// TIA Portal project "TPP" (V16)

(* hardware
DEVICE "S7300/ET200M station_1"  S7-300 station
   slot 0: "Rail_0"  Rail  6ES7 390-1***0-0AA0
   slot 2: "PLC_1"  CPU 314C-2 PN/DP  6ES7 314-6EH04-0AB0  V3.3
      slot 2: "PROFINET interface_1"  PN-IO
         slot 1: "Port_1"  Port
         slot 2: "Port_2"  Port
      slot 5: "DI 24/DO 16_1"  DI24/DO16
      slot 6: "AI 5/AO 2_1"  AI5/AO2
      slot 7: "Count_1"  Counter
      slot 8: "Positioning_1"  Positioning
DEVICE "HMI_1"  KTP1000 Basic color PN
   slot 0: "HMI_1"  KTP1000 Basic color PN  6AV6 647-0AF11-3AX0  12.0.0.0
   slot 1: "HMI_RT_1"  KTP1000 Basic color PN  6AV6 647-0AF11-3AX0  12.0.0.0
   slot 5: "HMI_1.IE_CP_1"  PROFINET Interface  12.0.0.0
      slot 1: "Interface PROFINET_1"  PROFINET Interface
         slot 1: "Port_1"  Port
*)

// ===== PLC "PLC_1"  CPU 314C-2 PN/DP =====

VAR_GLOBAL   // PLC tag table "Default tag table"
   "DE" AT %I0.1 : Bool;
   "PP" AT %I0.2 : Bool;
   "CS" AT %I0.3 : Bool;
   "AP" AT %I0.4 : Bool;
   "C1" AT %M3.7 : Bool;
   "C2" AT %M4.0 : Bool;
   "C3" AT %M4.1 : Bool;
   "C4" AT %M4.2 : Bool;
   "C5" AT %M4.3 : Bool;
   "C6" AT %M4.4 : Bool;
   "C7" AT %M4.5 : Bool;
   "C8" AT %M4.6 : Bool;
   "C9" AT %M4.7 : Bool;
   "C10" AT %M5.0 : Bool;
   "PA" AT %Q0.0 : Bool;
   "PV" AT %Q0.1 : Bool;
   "CV1" AT %Q0.2 : Bool;
   "CV2" AT %Q0.3 : Bool;
   "GA" AT %Q0.4 : Bool;
   "CPH" AT %Q0.5 : Bool;
   "CPL" AT %Q0.6 : Bool;
   "B1" AT %M0.0 : Bool;
   "B2" AT %M0.1 : Bool;
   "B3" AT %M0.2 : Bool;
   "B4" AT %M0.3 : Bool;
   "B5" AT %M0.4 : Bool;
   "B6" AT %M0.5 : Bool;
   "B7" AT %M0.6 : Bool;
   "B8" AT %M0.7 : Bool;
   "B9" AT %M1.0 : Bool;
   "B10" AT %M1.1 : Bool;
   "B11" AT %M1.2 : Bool;
   "B12" AT %M1.3 : Bool;
   "B13" AT %M1.4 : Bool;
   "B14" AT %M1.5 : Bool;
   "B15" AT %M1.6 : Bool;
   "B16" AT %M1.7 : Bool;
   "B17" AT %M2.0 : Bool;
   "B18" AT %M2.1 : Bool;
   "B19" AT %M2.2 : Bool;
   "T1" AT %M2.5 : Bool;
   "T2" AT %M2.6 : Bool;
   "T3" AT %M2.7 : Bool;
   "T4" AT %M3.0 : Bool;
   "T5" AT %M3.1 : Bool;
   "T6" AT %M3.2 : Bool;
   "T7" AT %M3.3 : Bool;
   "T8" AT %M3.4 : Bool;
   "T9" AT %M3.5 : Bool;
   "T10" AT %M3.6 : Bool;
   "T11" AT %M5.1 : Bool;
   "T12" AT %M5.2 : Bool;
   "T13" AT %M5.3 : Bool;
   "T14" AT %M5.4 : Bool;
   "H1" AT %I0.5 : Bool;
   "H2" AT %I0.6 : Bool;
   "H3" AT %I0.7 : Bool;
   "H4" AT %I1.0 : Bool;
   "H5" AT %I1.1 : Bool;
   "H6" AT %I1.2 : Bool;
   "L1" AT %I1.3 : Bool;
   "L2" AT %I1.4 : Bool;
   "S" AT %I1.5 : Bool;
   "TC" AT %I1.6 : Bool;
   "AA" AT %Q0.7 : Bool;
END_VAR

ORGANIZATION_BLOCK "Main"   // OB1, LAD
TITLE = "Main Program Sweep (Cycle)"
{ S7_Optimized_Access := 'FALSE' }
VERSION : 0.1
   VAR_TEMP
      OB1_EV_CLASS : Byte;   // Bits 0-3 = 1 (Coming event), Bits 4-7 = 1 (Event class 1)
      OB1_SCAN_1 : Byte;   // 1 (Cold restart scan 1 of OB 1), 3 (Scan 2-n of OB 1)
      OB1_PRIORITY : Byte;   // Priority of OB Execution
      OB1_OB_NUMBR : Byte;   // 1 (Organization block 1, OB1)
      OB1_RESERVED_1 : Byte;   // Reserved for system
      OB1_RESERVED_2 : Byte;   // Reserved for system
      OB1_PREV_CYCLE : Int;   // Cycle time of previous OB1 scan (milliseconds)
      OB1_MIN_CYCLE : Int;   // Minimum cycle time of OB1 (milliseconds)
      OB1_MAX_CYCLE : Int;   // Maximum cycle time of OB1 (milliseconds)
      OB1_DATE_TIME : Date_And_Time;   // Date and time OB1 started
   END_VAR
BEGIN

REGION Network 1
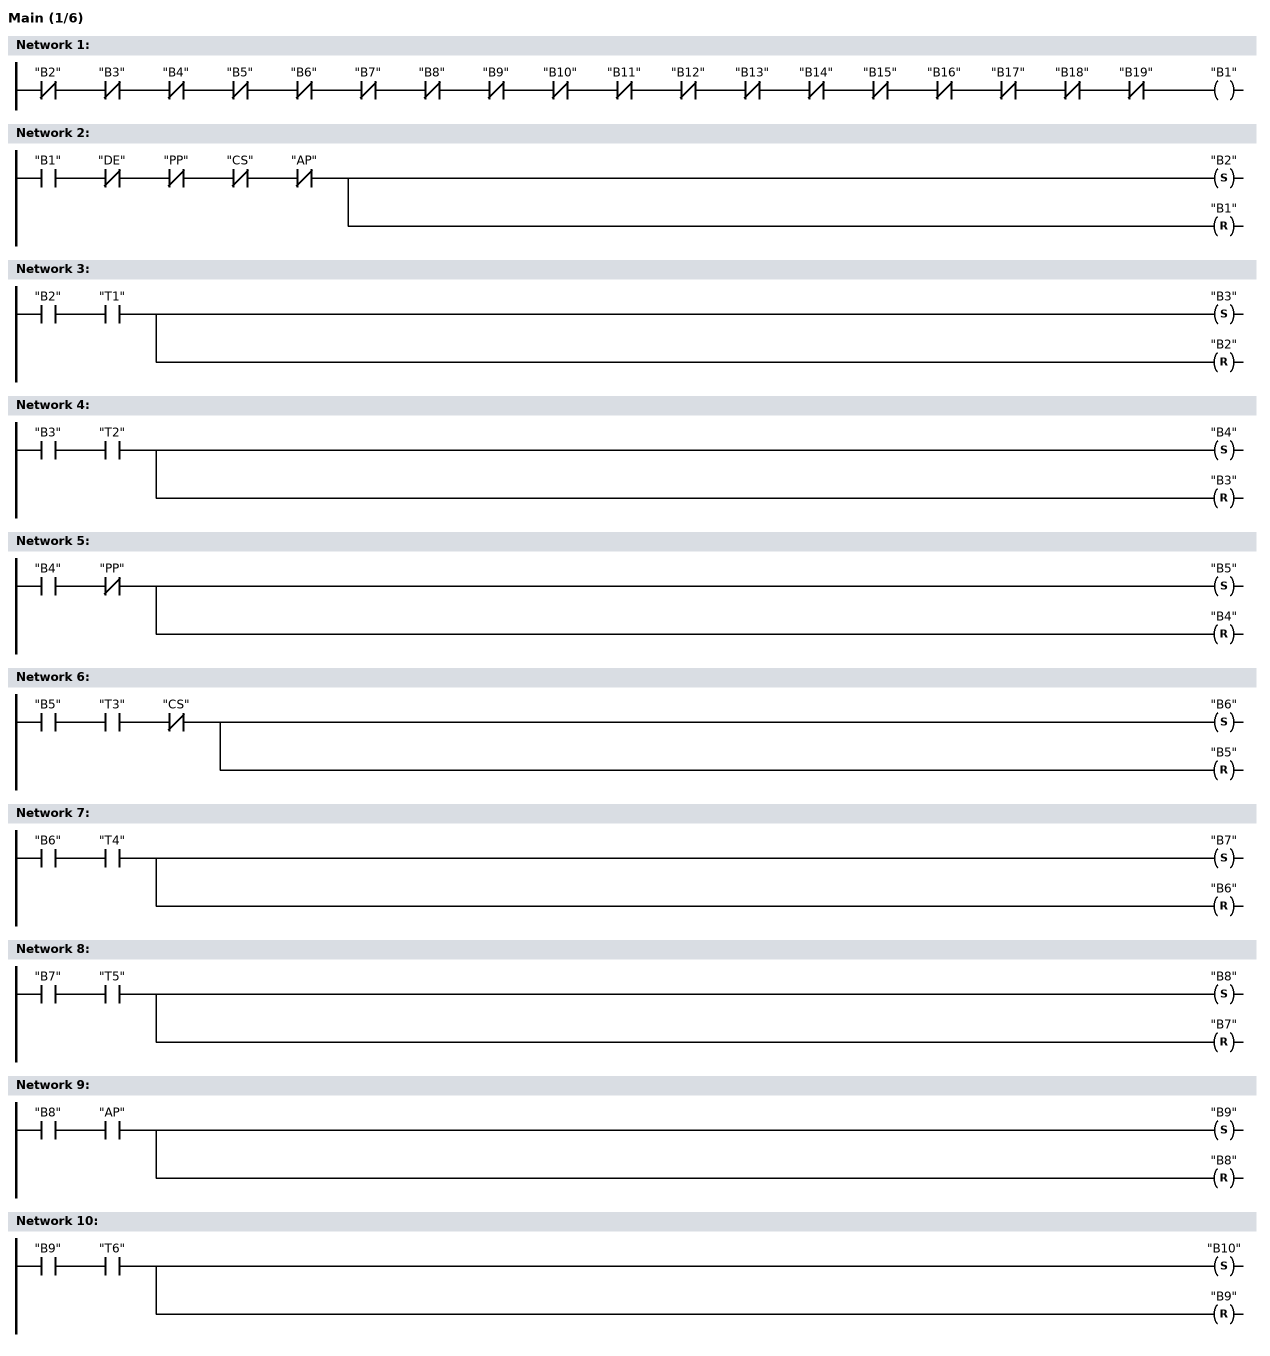
   RUNG wire#powerrail
      I_Contact( "B2" )
      I_Contact( "B3" )
      I_Contact( "B4" )
      I_Contact( "B5" )
      I_Contact( "B6" )
      I_Contact( "B7" )
      I_Contact( "B8" )
      I_Contact( "B9" )
      I_Contact( "B10" )
      I_Contact( "B11" )
      I_Contact( "B12" )
      I_Contact( "B13" )
      I_Contact( "B14" )
      I_Contact( "B15" )
      I_Contact( "B16" )
      I_Contact( "B17" )
      I_Contact( "B18" )
      I_Contact( "B19" )
      Coil( "B1" )
   END_RUNG
   // the same network as SCL:
   "B1" := NOT "B2" AND NOT "B3" AND NOT "B4" AND NOT "B5" AND NOT "B6" AND NOT "B7" AND NOT "B8" AND NOT "B9" AND NOT "B10" AND NOT "B11" AND NOT "B12" AND NOT "B13" AND NOT "B14" AND NOT "B15" AND NOT "B16" AND NOT "B17" AND NOT "B18" AND NOT "B19";
END_REGION

REGION Network 2
   RUNG wire#powerrail
      Contact( "B1" )
      I_Contact( "DE" )
      I_Contact( "PP" )
      I_Contact( "CS" )
      I_Contact( "AP" )
      wire#w1
      S_Coil( "B2" )
   END_RUNG
   RUNG wire#w1
      R_Coil( "B1" )
   END_RUNG
   // the same network as SCL:
   IF "B1" AND NOT "DE" AND NOT "PP" AND NOT "CS" AND NOT "AP" THEN
       "B2" := TRUE;
       "B1" := FALSE;
   END_IF;
END_REGION

REGION Network 3
   RUNG wire#powerrail
      Contact( "B2" )
      Contact( "T1" )
      wire#w1
      S_Coil( "B3" )
   END_RUNG
   RUNG wire#w1
      R_Coil( "B2" )
   END_RUNG
   // the same network as SCL:
   IF "B2" AND "T1" THEN
       "B3" := TRUE;
       "B2" := FALSE;
   END_IF;
END_REGION

REGION Network 4
   RUNG wire#powerrail
      Contact( "B3" )
      Contact( "T2" )
      wire#w1
      S_Coil( "B4" )
   END_RUNG
   RUNG wire#w1
      R_Coil( "B3" )
   END_RUNG
   // the same network as SCL:
   IF "B3" AND "T2" THEN
       "B4" := TRUE;
       "B3" := FALSE;
   END_IF;
END_REGION

REGION Network 5
   RUNG wire#powerrail
      Contact( "B4" )
      I_Contact( "PP" )
      wire#w1
      S_Coil( "B5" )
   END_RUNG
   RUNG wire#w1
      R_Coil( "B4" )
   END_RUNG
   // the same network as SCL:
   IF "B4" AND NOT "PP" THEN
       "B5" := TRUE;
       "B4" := FALSE;
   END_IF;
END_REGION

REGION Network 6
   RUNG wire#powerrail
      Contact( "B5" )
      Contact( "T3" )
      I_Contact( "CS" )
      wire#w1
      S_Coil( "B6" )
   END_RUNG
   RUNG wire#w1
      R_Coil( "B5" )
   END_RUNG
   // the same network as SCL:
   IF "B5" AND "T3" AND NOT "CS" THEN
       "B6" := TRUE;
       "B5" := FALSE;
   END_IF;
END_REGION

REGION Network 7
   RUNG wire#powerrail
      Contact( "B6" )
      Contact( "T4" )
      wire#w1
      S_Coil( "B7" )
   END_RUNG
   RUNG wire#w1
      R_Coil( "B6" )
   END_RUNG
   // the same network as SCL:
   IF "B6" AND "T4" THEN
       "B7" := TRUE;
       "B6" := FALSE;
   END_IF;
END_REGION

REGION Network 8
   RUNG wire#powerrail
      Contact( "B7" )
      Contact( "T5" )
      wire#w1
      S_Coil( "B8" )
   END_RUNG
   RUNG wire#w1
      R_Coil( "B7" )
   END_RUNG
   // the same network as SCL:
   IF "B7" AND "T5" THEN
       "B8" := TRUE;
       "B7" := FALSE;
   END_IF;
END_REGION

REGION Network 9
   RUNG wire#powerrail
      Contact( "B8" )
      Contact( "AP" )
      wire#w1
      S_Coil( "B9" )
   END_RUNG
   RUNG wire#w1
      R_Coil( "B8" )
   END_RUNG
   // the same network as SCL:
   IF "B8" AND "AP" THEN
       "B9" := TRUE;
       "B8" := FALSE;
   END_IF;
END_REGION

REGION Network 10
   RUNG wire#powerrail
      Contact( "B9" )
      Contact( "T6" )
      wire#w1
      S_Coil( "B10" )
   END_RUNG
   RUNG wire#w1
      R_Coil( "B9" )
   END_RUNG
   // the same network as SCL:
   IF "B9" AND "T6" THEN
       "B10" := TRUE;
       "B9" := FALSE;
   END_IF;
END_REGION

REGION Network 11
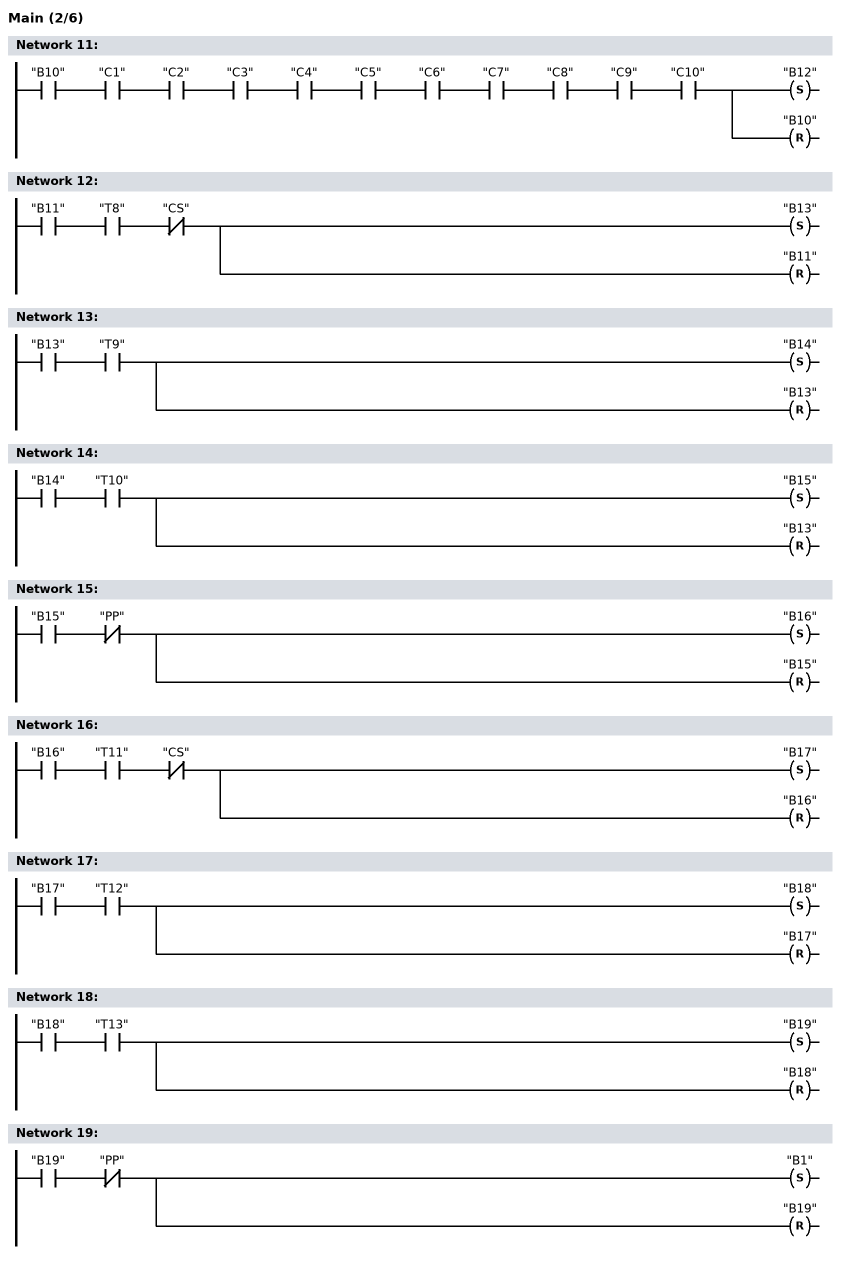
   RUNG wire#powerrail
      Contact( "B10" )
      Contact( "C1" )
      Contact( "C2" )
      Contact( "C3" )
      Contact( "C4" )
      Contact( "C5" )
      Contact( "C6" )
      Contact( "C7" )
      Contact( "C8" )
      Contact( "C9" )
      Contact( "C10" )
      wire#w1
      S_Coil( "B12" )
   END_RUNG
   RUNG wire#w1
      R_Coil( "B10" )
   END_RUNG
   // the same network as SCL:
   IF "B10" AND "C1" AND "C2" AND "C3" AND "C4" AND "C5" AND "C6" AND "C7" AND "C8" AND "C9" AND "C10" THEN
       "B12" := TRUE;
       "B10" := FALSE;
   END_IF;
END_REGION

REGION Network 12
   RUNG wire#powerrail
      Contact( "B11" )
      Contact( "T8" )
      I_Contact( "CS" )
      wire#w1
      S_Coil( "B13" )
   END_RUNG
   RUNG wire#w1
      R_Coil( "B11" )
   END_RUNG
   // the same network as SCL:
   IF "B11" AND "T8" AND NOT "CS" THEN
       "B13" := TRUE;
       "B11" := FALSE;
   END_IF;
END_REGION

REGION Network 13
   RUNG wire#powerrail
      Contact( "B13" )
      Contact( "T9" )
      wire#w1
      S_Coil( "B14" )
   END_RUNG
   RUNG wire#w1
      R_Coil( "B13" )
   END_RUNG
   // the same network as SCL:
   IF "B13" AND "T9" THEN
       "B14" := TRUE;
       "B13" := FALSE;
   END_IF;
END_REGION

REGION Network 14
   RUNG wire#powerrail
      Contact( "B14" )
      Contact( "T10" )
      wire#w1
      S_Coil( "B15" )
   END_RUNG
   RUNG wire#w1
      R_Coil( "B13" )
   END_RUNG
   // the same network as SCL:
   IF "B14" AND "T10" THEN
       "B15" := TRUE;
       "B13" := FALSE;
   END_IF;
END_REGION

REGION Network 15
   RUNG wire#powerrail
      Contact( "B15" )
      I_Contact( "PP" )
      wire#w1
      S_Coil( "B16" )
   END_RUNG
   RUNG wire#w1
      R_Coil( "B15" )
   END_RUNG
   // the same network as SCL:
   IF "B15" AND NOT "PP" THEN
       "B16" := TRUE;
       "B15" := FALSE;
   END_IF;
END_REGION

REGION Network 16
   RUNG wire#powerrail
      Contact( "B16" )
      Contact( "T11" )
      I_Contact( "CS" )
      wire#w1
      S_Coil( "B17" )
   END_RUNG
   RUNG wire#w1
      R_Coil( "B16" )
   END_RUNG
   // the same network as SCL:
   IF "B16" AND "T11" AND NOT "CS" THEN
       "B17" := TRUE;
       "B16" := FALSE;
   END_IF;
END_REGION

REGION Network 17
   RUNG wire#powerrail
      Contact( "B17" )
      Contact( "T12" )
      wire#w1
      S_Coil( "B18" )
   END_RUNG
   RUNG wire#w1
      R_Coil( "B17" )
   END_RUNG
   // the same network as SCL:
   IF "B17" AND "T12" THEN
       "B18" := TRUE;
       "B17" := FALSE;
   END_IF;
END_REGION

REGION Network 18
   RUNG wire#powerrail
      Contact( "B18" )
      Contact( "T13" )
      wire#w1
      S_Coil( "B19" )
   END_RUNG
   RUNG wire#w1
      R_Coil( "B18" )
   END_RUNG
   // the same network as SCL:
   IF "B18" AND "T13" THEN
       "B19" := TRUE;
       "B18" := FALSE;
   END_IF;
END_REGION

REGION Network 19
   RUNG wire#powerrail
      Contact( "B19" )
      I_Contact( "PP" )
      wire#w1
      S_Coil( "B1" )
   END_RUNG
   RUNG wire#w1
      R_Coil( "B19" )
   END_RUNG
   // the same network as SCL:
   IF "B19" AND NOT "PP" THEN
       "B1" := TRUE;
       "B19" := FALSE;
   END_IF;
END_REGION

REGION Network 20
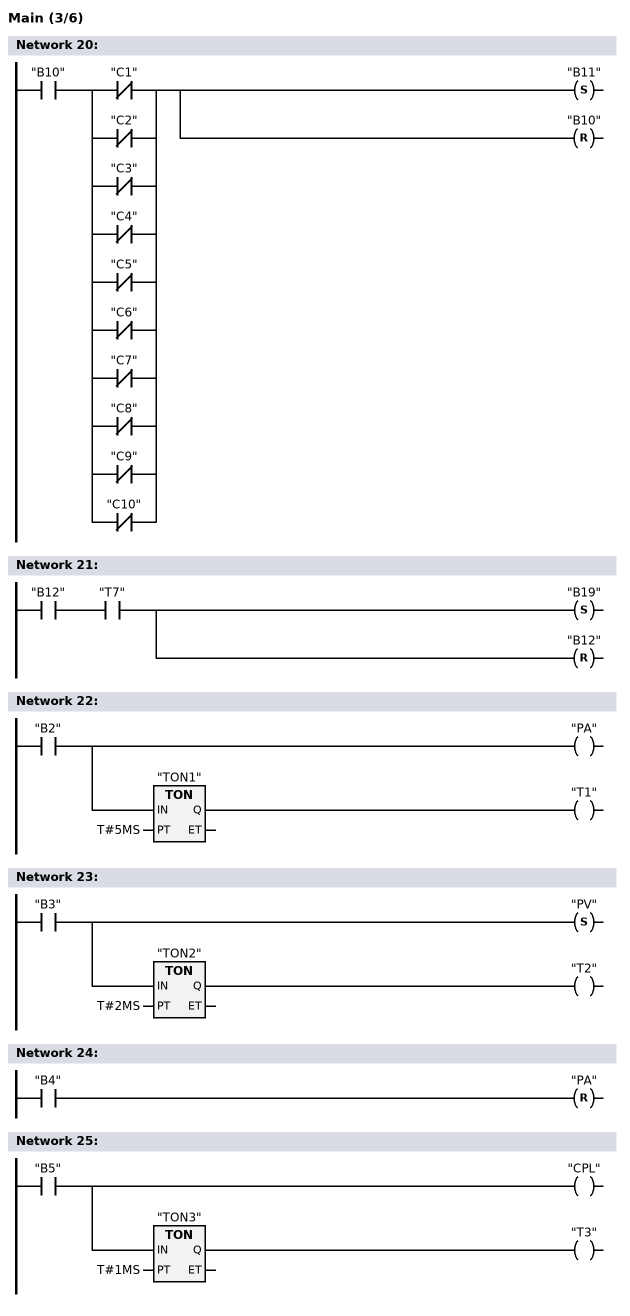
   RUNG wire#powerrail
      Contact( "B10" )
      wire#w1
      I_Contact( "C1" )
      wire#w2
      S_Coil( "B11" )
   END_RUNG
   RUNG wire#w1
      I_Contact( "C2" )
   END_RUNG wire#w2
   RUNG wire#w1
      I_Contact( "C3" )
   END_RUNG wire#w2
   RUNG wire#w1
      I_Contact( "C4" )
   END_RUNG wire#w2
   RUNG wire#w1
      I_Contact( "C5" )
   END_RUNG wire#w2
   RUNG wire#w1
      I_Contact( "C6" )
   END_RUNG wire#w2
   RUNG wire#w1
      I_Contact( "C7" )
   END_RUNG wire#w2
   RUNG wire#w1
      I_Contact( "C8" )
   END_RUNG wire#w2
   RUNG wire#w1
      I_Contact( "C9" )
   END_RUNG wire#w2
   RUNG wire#w1
      I_Contact( "C10" )
   END_RUNG wire#w2
   RUNG wire#w2
      R_Coil( "B10" )
   END_RUNG
   // the same network as SCL:
   IF "B10" AND (NOT "C1" OR NOT "C2" OR NOT "C3" OR NOT "C4" OR NOT "C5" OR NOT "C6" OR NOT "C7" OR NOT "C8" OR NOT "C9" OR NOT "C10") THEN
       "B11" := TRUE;
       "B10" := FALSE;
   END_IF;
END_REGION

REGION Network 21
   RUNG wire#powerrail
      Contact( "B12" )
      Contact( "T7" )
      wire#w1
      S_Coil( "B19" )
   END_RUNG
   RUNG wire#w1
      R_Coil( "B12" )
   END_RUNG
   // the same network as SCL:
   IF "B12" AND "T7" THEN
       "B19" := TRUE;
       "B12" := FALSE;
   END_IF;
END_REGION

REGION Network 22
   "PA" := "B2";
   "TON1".TON(IN := "B2", PT := T#5MS);
   "T1" := "TON1".Q;
END_REGION

REGION Network 23
   IF "B3" THEN "PV" := TRUE; END_IF;
   "TON2".TON(IN := "B3", PT := T#2MS);
   "T2" := "TON2".Q;
END_REGION

REGION Network 24
   RUNG wire#powerrail
      Contact( "B4" )
      R_Coil( "PA" )
   END_RUNG
   // the same network as SCL:
   IF "B4" THEN "PA" := FALSE; END_IF;
END_REGION

REGION Network 25
   "CPL" := "B5";
   "TON3".TON(IN := "B5", PT := T#1MS);
   "T3" := "TON3".Q;
END_REGION

REGION Network 26
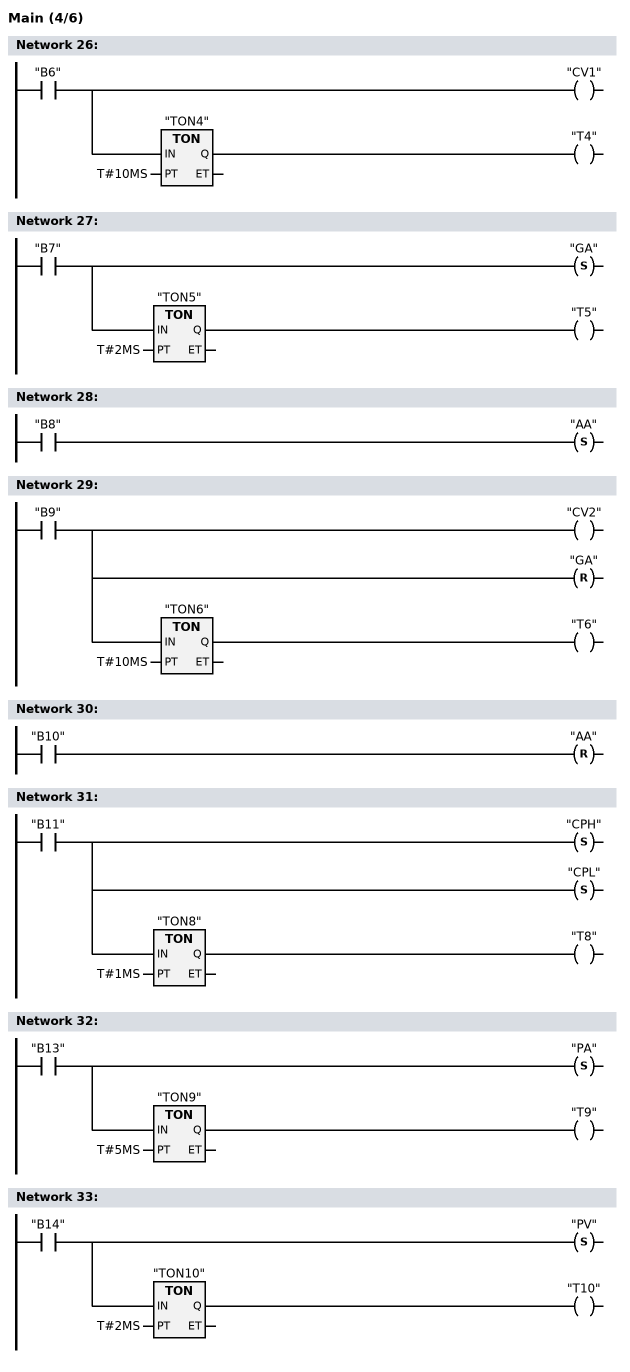
   "CV1" := "B6";
   "TON4".TON(IN := "B6", PT := T#10MS);
   "T4" := "TON4".Q;
END_REGION

REGION Network 27
   IF "B7" THEN "GA" := TRUE; END_IF;
   "TON5".TON(IN := "B7", PT := T#2MS);
   "T5" := "TON5".Q;
END_REGION

REGION Network 28
   RUNG wire#powerrail
      Contact( "B8" )
      S_Coil( "AA" )
   END_RUNG
   // the same network as SCL:
   IF "B8" THEN "AA" := TRUE; END_IF;
END_REGION

REGION Network 29
   "CV2" := "B9";
   IF "B9" THEN "GA" := FALSE; END_IF;
   "TON6".TON(IN := "B9", PT := T#10MS);
   "T6" := "TON6".Q;
END_REGION

REGION Network 30
   RUNG wire#powerrail
      Contact( "B10" )
      R_Coil( "AA" )
   END_RUNG
   // the same network as SCL:
   IF "B10" THEN "AA" := FALSE; END_IF;
END_REGION

REGION Network 31
   IF "B11" THEN
       "CPH" := TRUE;
       "CPL" := TRUE;
   END_IF;
   "TON8".TON(IN := "B11", PT := T#1MS);
   "T8" := "TON8".Q;
END_REGION

REGION Network 32
   IF "B13" THEN "PA" := TRUE; END_IF;
   "TON9".TON(IN := "B13", PT := T#5MS);
   "T9" := "TON9".Q;
END_REGION

REGION Network 33
   IF "B14" THEN "PV" := TRUE; END_IF;
   "TON10".TON(IN := "B14", PT := T#2MS);
   "T10" := "TON10".Q;
END_REGION

REGION Network 34
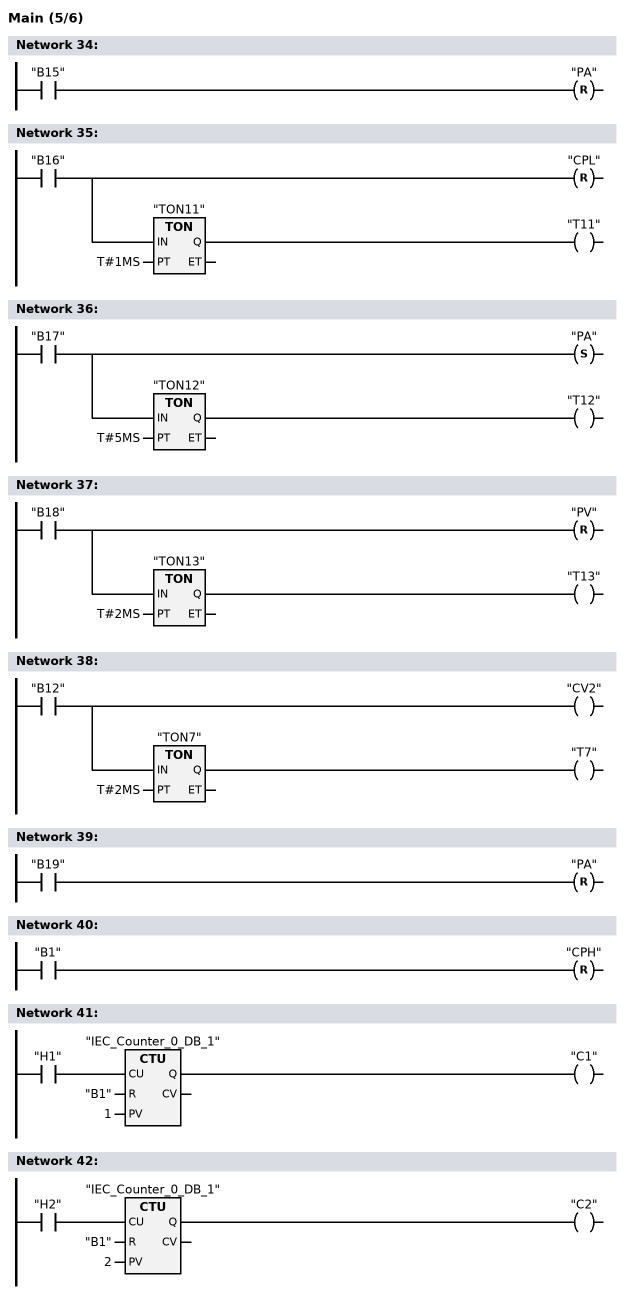
   RUNG wire#powerrail
      Contact( "B15" )
      R_Coil( "PA" )
   END_RUNG
   // the same network as SCL:
   IF "B15" THEN "PA" := FALSE; END_IF;
END_REGION

REGION Network 35
   IF "B16" THEN "CPL" := FALSE; END_IF;
   "TON11".TON(IN := "B16", PT := T#1MS);
   "T11" := "TON11".Q;
END_REGION

REGION Network 36
   IF "B17" THEN "PA" := TRUE; END_IF;
   "TON12".TON(IN := "B17", PT := T#5MS);
   "T12" := "TON12".Q;
END_REGION

REGION Network 37
   IF "B18" THEN "PV" := FALSE; END_IF;
   "TON13".TON(IN := "B18", PT := T#2MS);
   "T13" := "TON13".Q;
END_REGION

REGION Network 38
   "CV2" := "B12";
   "TON7".TON(IN := "B12", PT := T#2MS);
   "T7" := "TON7".Q;
END_REGION

REGION Network 39
   RUNG wire#powerrail
      Contact( "B19" )
      R_Coil( "PA" )
   END_RUNG
   // the same network as SCL:
   IF "B19" THEN "PA" := FALSE; END_IF;
END_REGION

REGION Network 40
   RUNG wire#powerrail
      Contact( "B1" )
      R_Coil( "CPH" )
   END_RUNG
   // the same network as SCL:
   IF "B1" THEN "CPH" := FALSE; END_IF;
END_REGION

REGION Network 41
   "IEC_Counter_0_DB_1".CTU(CU := "H1", R := "B1", PV := 1);
   "C1" := "IEC_Counter_0_DB_1".Q;
END_REGION

REGION Network 42
   "IEC_Counter_0_DB_1".CTU(CU := "H2", R := "B1", PV := 2);
   "C2" := "IEC_Counter_0_DB_1".Q;
END_REGION

REGION Network 43
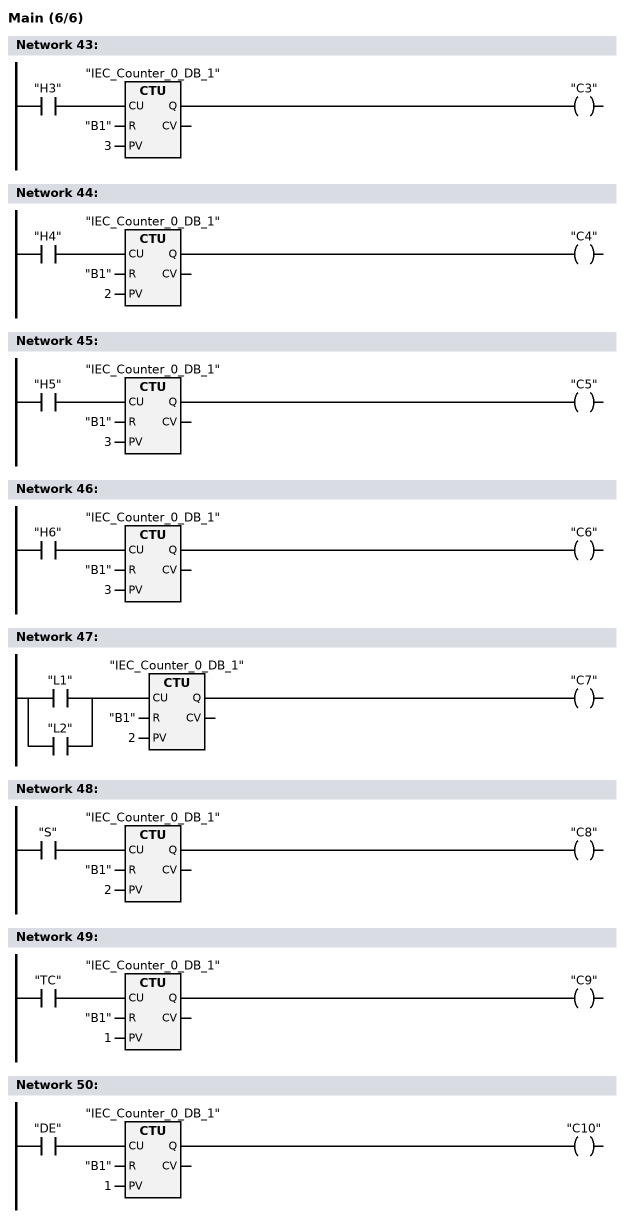
   "IEC_Counter_0_DB_1".CTU(CU := "H3", R := "B1", PV := 3);
   "C3" := "IEC_Counter_0_DB_1".Q;
END_REGION

REGION Network 44
   "IEC_Counter_0_DB_1".CTU(CU := "H4", R := "B1", PV := 2);
   "C4" := "IEC_Counter_0_DB_1".Q;
END_REGION

REGION Network 45
   "IEC_Counter_0_DB_1".CTU(CU := "H5", R := "B1", PV := 3);
   "C5" := "IEC_Counter_0_DB_1".Q;
END_REGION

REGION Network 46
   "IEC_Counter_0_DB_1".CTU(CU := "H6", R := "B1", PV := 3);
   "C6" := "IEC_Counter_0_DB_1".Q;
END_REGION

REGION Network 47
   "IEC_Counter_0_DB_1".CTU(CU := "L1" OR "L2", R := "B1", PV := 2);
   "C7" := "IEC_Counter_0_DB_1".Q;
END_REGION

REGION Network 48
   "IEC_Counter_0_DB_1".CTU(CU := "S", R := "B1", PV := 2);
   "C8" := "IEC_Counter_0_DB_1".Q;
END_REGION

REGION Network 49
   "IEC_Counter_0_DB_1".CTU(CU := "TC", R := "B1", PV := 1);
   "C9" := "IEC_Counter_0_DB_1".Q;
END_REGION

REGION Network 50
   "IEC_Counter_0_DB_1".CTU(CU := "DE", R := "B1", PV := 1);
   "C10" := "IEC_Counter_0_DB_1".Q;
END_REGION
END_ORGANIZATION_BLOCK

(* ===== HMI "HMI_RT_1" =====
system functions are stored by id; their names below are inferred from use
connection "HMI_Liaison_1": ETHERNET, SIMATIC S7 300/400 MPI

HMI tags "Table de variables standard"
   "Numéro_vue_variable" : UInt, internal
   "DE" : Bool = PLC DE AT %I0.1, 1 s
   "move" : Int, internal
   "PP" : Bool = PLC PP AT %I0.2, 1 s
   "S" : Bool = PLC S AT %I1.5, 1 s
   "TC" : Bool = PLC TC AT %I1.6, 1 s
   "L1" : Bool = PLC L1 AT %I1.3, 1 s
   "L2" : Bool = PLC L2 AT %I1.4, 1 s
   "H1" : Bool = PLC H1 AT %I0.5, 1 s
   "H2" : Bool = PLC H2 AT %I0.6, 1 s
   "H3" : Bool = PLC H3 AT %I0.7, 1 s
   "H4" : Bool = PLC H4 AT %I1.0, 1 s
   "H5" : Bool = PLC H5 AT %I1.1, 1 s
   "H6" : Bool = PLC H6 AT %I1.2, 1 s

Template "Modèle_1" 640x480
   Button "Exit" at 560,422 size 79x57; TextOff 'Exit'; PictureOff "ExitRuntime_KTP1000_Basic_color_PN"; PictureOn "ExitRuntime_KTP1000_Basic_color_PN"
      on Release: StopRuntime(0)
   Button "Template_Button" at 480,422 size 79x57; TextOff 'Text'
   Button "Template_Button_1" at 400,422 size 79x57; TextOff 'Text'
   Button "Template_Button_2" at 320,422 size 79x57; TextOff 'Text'
   Button "Template_Button_3" at 240,422 size 79x57; TextOff 'Text'
   Button "Template_Button_4" at 160,422 size 79x57; TextOff 'Text'
   Button "Alarms" at 80,422 size 79x57; TextOff 'Alarms'; PictureOff "AlarmDisplay_KTP1000_Basic_color_PN"; PictureOn "AlarmDisplay_KTP1000_Basic_color_PN"
      on Release: function_ef3f5d25("Fenêtre des alarmes_non acquittée", -1)
   Button "Start screen" at 0,422 size 79x57; TextOff 'Start screen'; PictureOff "NavigateHome_KTP1000_Basic_color_PN"; PictureOn "NavigateHome_KTP1000_Basic_color_PN"
      on Release: ActivateScreen("Vue racine", 0)
   SymbolicIOField "Vue_champ_ES_symbolique" at 105,11 size 428x34; TextOff '0'; TextOn '1'; TextList "TextList_ScreenNames"
      ProcessValue <- "Numéro_vue_variable"
      on Change: ActivateScreenByNumber("Numéro_vue_variable", 0)
   DateTimeField "HmiScreenItemData" at 535,29 size 105x29
   DateTimeField "HmiScreenItemData_1" at 535,0 size 105x29
   GraphicView "Logo" at 0,0 size 103x58; Picture "Logo of HMI_1"

screen "Vue racine" 640x480, template "Modèle_1"
   on GenerateScreen: SetTag("Numéro_vue_variable", 1); function_f9c01323("move", 1, 100, 0, 1)
   GraphicView "Graphic view_21" at 236,57 size 40x96; Picture "Graphic_5"
      VerticalMovement <- "move"
      Visibility <- "PP"
   GraphicView "Graphic view_6" at 77,173 size 201x132; Picture "Graphic_4"
   GraphicView "Graphic view_5" at 276,201 size 201x132; Picture "Graphic_4"
   GraphicView "Graphic view_15" at 320,67 size 48x86; Picture "Graphic_5"
   GraphicView "Graphic view_20" at 175,59 size 48x86; Picture "Graphic_5"
   GraphicView "Graphic view_8" at 440,79 size 48x86; Picture "Graphic_5"
   GraphicView "Graphic view_3" at 130,102 size 29x39; Picture "Graphique_6"
   GraphicView "Graphic view_1" at 25,279 size 52x32; Picture "Graphic_1"
   Button "Button_1" at 104,82 size 26x20; TextOff 'DE'
      on Press: SetBit("DE")
      Appearance <- "DE"
   GraphicView "Graphic view_11" at 236,199 size 29x39; Picture "Graphique_6"
   GraphicView "Graphic view_13" at 364,280 size 29x39; Picture "Graphique_6"
   GraphicView "Graphic view_14" at 95,216 size 29x39; Picture "Graphique_6"
   Button "Button_3" at 498,231 size 26x20; TextOff 'L1'
      on Press: SetBit("L1")
      Appearance <- "L1"
   Button "Button_4" at 393,303 size 26x21; TextOff 'H5'
      on Press: SetBit("H5")
      Appearance <- "H5"
   Button "Button_5" at 64,238 size 26x20; TextOff 'S'
      on Press: SetBit("S")
      Appearance <- "S"
   Button "Button_6" at 267,207 size 19x20; TextOff 'T'
      on Press: SetBit("TC")
      Appearance <- "TC"
   GraphicView "Graphic view_12" at 461,207 size 29x39; Picture "Graphique_6"
   GraphicView "Graphic view_22" at 430,141 size 56x65; Picture "Graphic_6"
   GraphicView "Graphic view_4" at 316,132 size 56x65; Picture "Graphic_6"
   GraphicView "Graphic view_7" at 167,120 size 56x65; Picture "Graphic_6"
   GraphicView "Graphic view_25" at 92,283 size 98x73; Picture "Graphic_10"
   GraphicView "Graphic view_2" at 219,305 size 55x38; Picture "Graphic_1"
   GraphicView "Graphic view_9" at 379,183 size 29x39; Picture "Graphique_6"
   Button "Button_2" at 358,207 size 26x20; TextOff 'L2'
      on Press: SetBit("L2")
      Appearance <- "L2"
   GraphicView "Graphic view_10" at 343,303 size 29x39; Picture "Graphique_6"
   GraphicView "Graphic view_16" at 401,258 size 29x39; Picture "Graphique_6"
   GraphicView "Graphic view_17" at 247,266 size 29x39; Picture "Graphique_6"
   GraphicView "Graphic view_18" at 278,251 size 29x39; Picture "Graphique_6"
   GraphicView "Graphic view_19" at 316,231 size 29x39; Picture "Graphique_6"
   Button "Button_7" at 362,324 size 26x21; TextOff 'H4'
      on Press: SetBit("H4")
      Appearance <- "H4"
   Button "Button_8" at 320,253 size 28x19; TextOff 'H3'
      on Press: SetBit("H3")
      Appearance <- "H3"
   Button "Button_9" at 262,298 size 24x21; TextOff 'H1'
      on Press: SetBit("H1")
      Appearance <- "H1"
   Button "Button_10" at 288,270 size 25x22; TextOff 'H2'
      on Press: SetBit("H2")
      Appearance <- "H2"
   Button "Button_11" at 425,272 size 26x20; TextOff 'H6'
      on Press: SetBit("H6")
      Appearance <- "H6"
*)